Fanuc KAREL source: kb00123.KL

-- PROVISIONAL review KL for V770-1; original PC SHA256 9a30d74417f775517e5523e04ec991e03dbc85cdfa3ef1b8afddc7cfb8125376
-- Incomplete behavior may be omitted. Consult companion uncertainty JSON. Do not deploy.
PROGRAM KB00123
%NOLOCKGROUP
BEGIN
  -- UNRESOLVED_PC offsets 5-14; opcodes 3F,75
  -- UNRESOLVED_PC offsets 19-26; opcodes 9D,23
  -- UNRESOLVED_PC offsets 31-49; opcodes 27,22,2A,22,31
  -- UNRESOLVED_PC offsets 54-58; opcodes 7F
END KB00123
